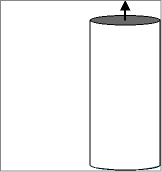
VISUALIZATION VISU_Tube_Top_14  // 162x172
VAR_IN_OUT
	azi : LREAL;
END_VAR
    Ellipse (90,160 70x10)
        p2858320360: azi
    Polygon (90,20) (160,20) (160,165) (152,167) (146,168) (138,169) (131,169) (123,169) (114,169) (104,168) (95,167) (90,165)
        p2858320360: azi
    Ellipse (90,15 70x10)
        p2858320360: azi
    Polygon (120,10) (125,0) (130,10)
        p2858320360: azi
    Polyline (125,20) (125,10)
        p2858320360: azi
    Polyline (160,165) (160,20)
        p2858320360: azi
    Polyline (90,165) (90,20)
        p2858320360: azi
END_VISUALIZATION

(* stored: Version 1.1.0.1, ProductVersion 3.1.4018.5
   Visu VISU_Tube_Top_14: Id {b5788192-feac-459c-8ba2-047074780a33} *)
